FUNCTION_BLOCK FB_RunHOMSWithBender EXTENDS FB_RunHOMS
VAR_INPUT
END_VAR
VAR_OUTPUT
END_VAR
VAR_IN_OUT
    stYup : DUT_MotionStage;
    stYdwn : DUT_MotionStage;
    stXup : DUT_MotionStage;
    stXdwn : DUT_MotionStage;
    stPitch : DUT_MotionStage;
    stBender : DUT_MotionStage;

    bExecuteCoupleY : BOOL;
    bExecuteCoupleX : BOOL;
    bExecuteDecoupleY : BOOL;
    bExecuteDecoupleX : BOOL;
END_VAR
VAR
END_VAR

SUPER^(stYup:=stYup,
       stYdwn:=stYdwn,
       stXup:=stXup,
       stXdwn:=stXdwn,
       stPitch:=stPitch,
       bExecuteCoupleY:=bExecuteCoupleY,
       bExecuteCoupleX:=bExecuteCoupleX,
       bExecuteDecoupleY:=bExecuteDecoupleY,
       bExecuteDecoupleX:=bExecuteDecoupleX);
stBender.bHardwareEnable := bSTOEnable1 AND bSTOEnable2;

END_FUNCTION_BLOCK

(* stored: Version 1.1.0.1, ProductVersion 3.1.4022.18
   POU FB_RunHOMSWithBender: Id {5da7a337-7cbf-48fc-8f67-1355602efa04}, SpecialFunc None *)
